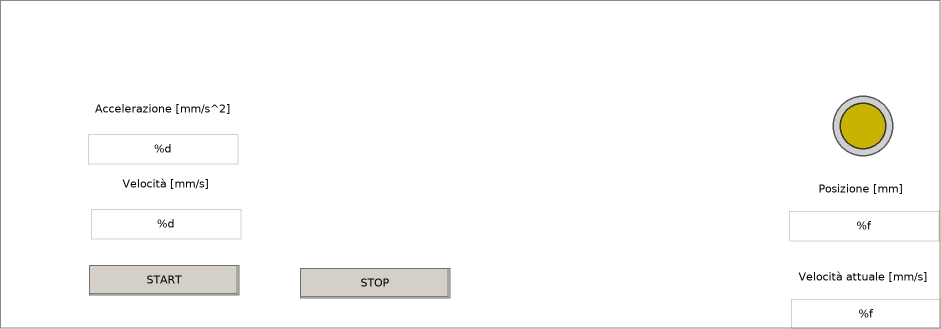
VISUALIZATION Visualization  // 941x329
    Lamp1 (828,91 70x70), variable: GVL.bMotorForward, style: Lamp-Lamp1-Yellow
    Button (89,265 150x30), "START"
        tap GVL.bStartButton
    Button (300,268 150x30), "STOP"
        tap GVL.bStopButton
    Textfield (789,211 150x30), "%f", text variable: GVL.nMotorPosition
    Textfield (91,209 150x30), "%d", text variable: GVL.fVelocity
        OnMouseClick: write the text variable via Default, min 0, max 7000, title "Velocità"
    Label (91,169 150x30), "Velocità [mm/s]"
    Label (786,174 150x30), "Posizione [mm]"
    Textfield (791,299 150x30), "%f", text variable: GVL.axis.NcToPlc.ActVelo
    Label (788,262 150x30), "Velocità attuale [mm/s]"
    Textfield (88,134 150x30), "%d", text variable: GVL.fAccelleration
        OnMouseClick: write the text variable via Default, min 0, max 500, title "Velocità"
    Label (88,94 150x30), "Accelerazione [mm/s^2]"
END_VISUALIZATION

(* stored: Version 1.1.0.1, ProductVersion 3.1.4024.12
   Visu Visualization: Id {8307b292-c0ff-42ce-a616-db2f7f9ed27b} *)
